(* Schneider Machine Expert - Basic project p12, file version 1.8.0.0 *)
(* ProjectInformations: Name=New project *)

HARDWARE
  Cpu 0: TM221CE16R
  EthernetConfiguration: NetworkName=M221, IpAllocationMode=FixedAddress, IpAddress=192.168.162.202, SubnetMask=255.255.255.0
  SerialLineConfiguration: Baud=Baud19200, Parity=ParityEven, DataBits=DataBits8, StopBits=StopBits1, PhysicalMedium=PhysicalMediumRs485, TransmissionMode=TransmissionModeModbusRtu, SlaveId=1, Addressing=SlaveAddressing
  MastTask: UsePeriodScanMode=false, PeriodScan=100
  FastTask: Period=255
  CpuBehavior: StartingMode=StartAsPreviousState, AutoSaveRamOnEeprom=true, WatchdogPeriod=250

SYMBOLS  (address, symbol, comment, settings)
  %C0         [Preset=5]

POU New POU
  (* SectionNumber=1 *)

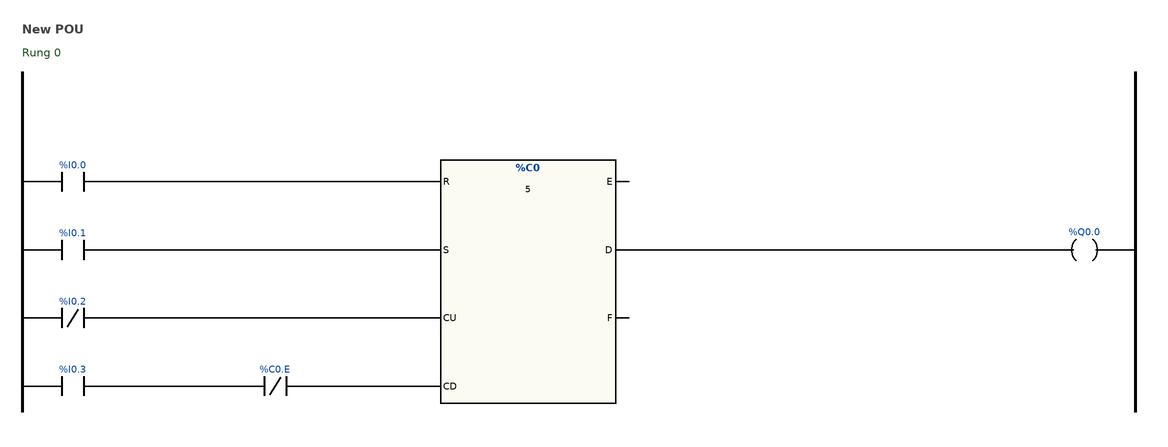

// Rung 0
  BLK %C0
  LD %I0.0
  R
  LD %I0.1
  S
  LDN %I0.2
  CU
  LD %I0.3
  ANDN %C0.E
  CD
  OUT_BLK
  LD D
  ST %Q0.0
  END_BLK
  // as ST:
  //   %C0(R := %I0.0, S := %I0.1, CU := NOT %I0.2, CD := %I0.3 AND NOT %C0.E);
  //   %Q0.0 := %C0.D;
